{attribute 'no_explicit_call' := 'do not call this FB directly'}{attribute 'enable_dynamic_creation'}
FUNCTION_BLOCK FINAL BooleanDisplayNode EXTENDS Node
VAR
	in : _BOOL(FALSE);
	display : _BOOL(FALSE);
END_VAR

METHOD PUBLIC Clone : I_Node
VAR
	pNode : POINTER TO BooleanDisplayNode;
END_VAR
pNode := __NEW(BooleanDisplayNode);
Clone := pNode^;
END_METHOD

METHOD FB_init : BOOL
VAR_INPUT
	bInitRetains : BOOL; // if TRUE, the retain variables are initialized (warm start / cold start)
	bInCopyCode : BOOL;  // if TRUE, the instance afterwards gets moved into the copy code (online change)
END_VAR
AddInput('in', in);
AddContent('display', display);
END_METHOD

METHOD PROTECTED OnExecute : HRESULT
display.Value := in.Value;
END_METHOD

END_FUNCTION_BLOCK

(* stored: Version 1.1.0.1, ProductVersion 3.1.4024.12
   POU BooleanDisplayNode: Id {198c7521-1e12-0d04-01d4-91e52ee4f612}, SpecialFunc None
   Folder Constructor: Id {8761cb93-b94b-473f-9272-e99159b5e081}
   Method Clone: Id {fe15fbb0-95d8-43e8-9272-57a633d25d58}
   Method FB_init: Id {fdebc071-57d9-4545-9e95-e3651aa87bbe}
   Method OnExecute: Id {3eea65a5-6bf3-0e0b-2473-3b373deefdf4} *)
